PROGRAM SLL
VAR_INPUT
	SteadyStateRegion	:REAL;
END_VAR
VAR_OUTPUT
	ControllerOn		:BOOL;
	ControllerSwitch	:BOOL;
END_VAR
VAR
	u2b			:fbU2B;
	b2u			:fbB2U;
	split1		:fbSplit;
	split2		:fbSplit;
	r_trigu		:R_TRIG;
	r_trigd		:R_TRIG;
	IfElse1		:fbIfElse;
	IfElse2		:fbIfElse;
END_VAR
VAR // added by the converter: edge detectors and wires of the graphical bodies
    _w1, _w2 : BOOL;
    _w3 : ANY;
END_VAR


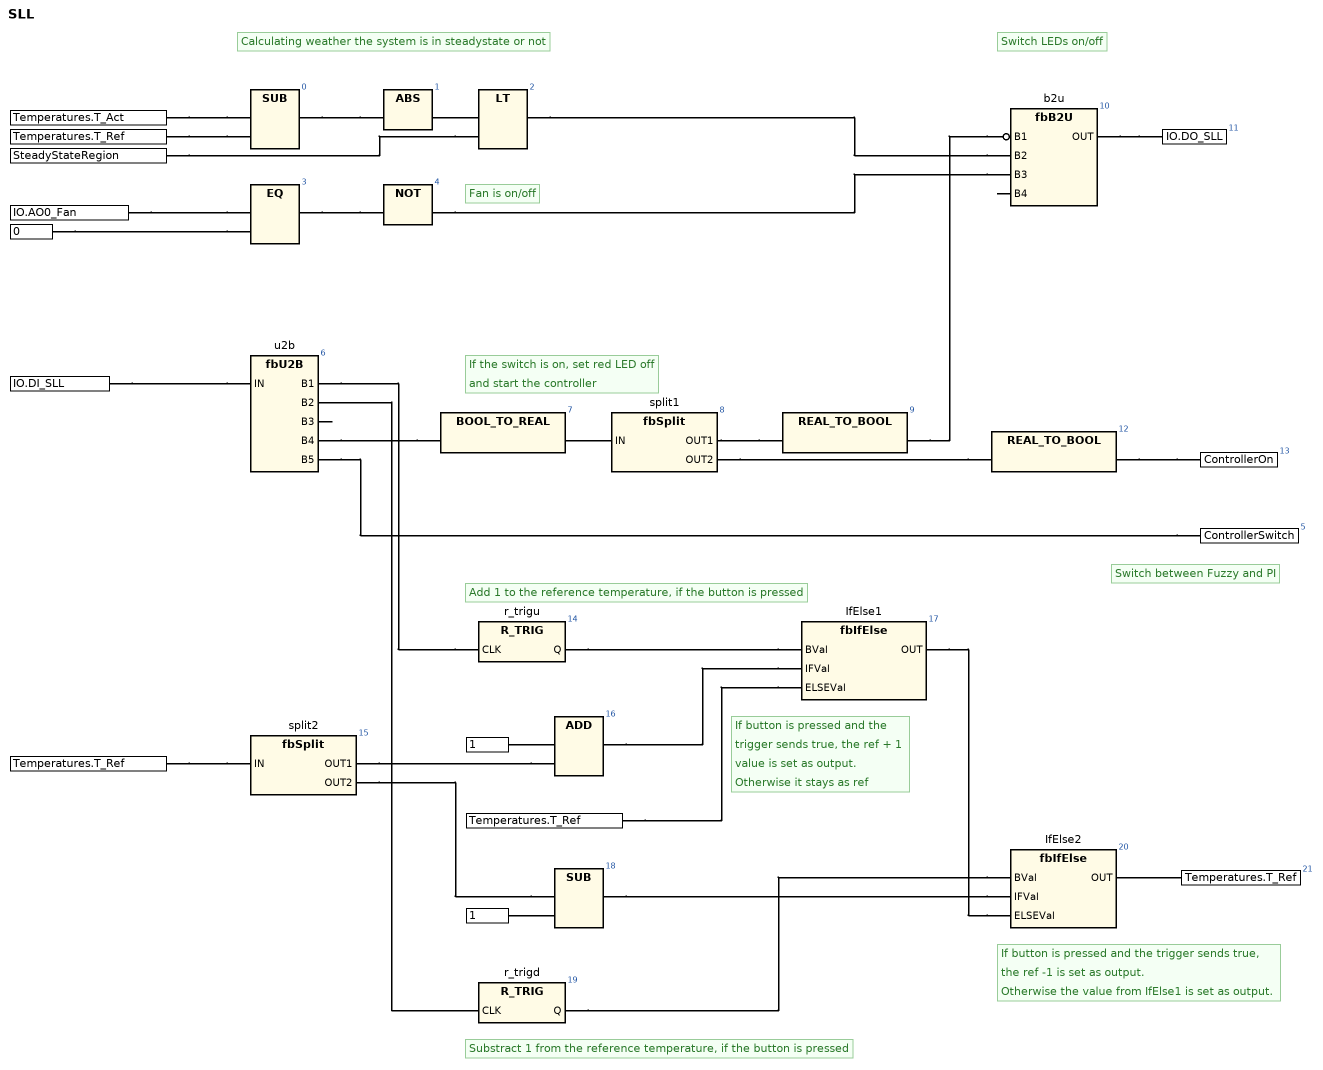
// PAGE -1
// Calculating weather the system is in steadystate or not
_w1 := ABS(Temperatures.T_Act - Temperatures.T_Ref) < SteadyStateRegion;
// Fan is on/off
_w2 := NOT (IO.AO0_Fan = 0);
// Switch between Fuzzy and PI
ControllerSwitch := u2b.B5;
u2b(IN := IO.DI_SLL); // fbU2B
// If the switch is on, set red LED off
// and start the controller
split1(IN := BOOL_TO_REAL(u2b.B4)); // fbSplit
// Switch LEDs on/off
b2u(B1 := NOT REAL_TO_BOOL(split1.OUT1), B2 := _w1, B3 := _w2); // fbB2U
IO.DO_SLL := b2u.OUT;
ControllerOn := REAL_TO_BOOL(split1.OUT2);
// Add 1 to the reference temperature, if the button is pressed
r_trigu(CLK := u2b.B1); // R_TRIG
split2(IN := Temperatures.T_Ref); // fbSplit
// If button is pressed and the
// trigger sends true, the ref + 1
// value is set as output.
// Otherwise it stays as ref
IfElse1(BVal := r_trigu.Q, IFVal := 1 + split2.OUT1, ELSEVal := Temperatures.T_Ref); // fbIfElse
_w3 := split2.OUT2 - 1;
// If button is pressed and the trigger sends true,
// the ref -1 is set as output.
// Otherwise the value from IfElse1 is set as output.
// Substract 1 from the reference temperature, if the button is pressed
r_trigd(CLK := u2b.B2); // R_TRIG
IfElse2(BVal := r_trigd.Q, IFVal := _w3, ELSEVal := IfElse1.OUT); // fbIfElse
Temperatures.T_Ref := IfElse2.OUT;

END_PROGRAM

(* stored: Version 1.1.0.1, ProductVersion 3.1.4022.6
   POU SLL: Id {4549d1e5-0425-4dde-8121-2f8eee1d555f}, SpecialFunc None *)
